FUNCTION FUN_InsideHysteresis : BOOL
VAR_INPUT
	rAct		:LREAL;			// Actual value
	rSp			:LREAL;			// Setpoint value
	rHys		:LREAL;			// Hysteresis	
END_VAR
VAR
	bInside		:BOOL;			// True if actual value is within setpoint plus minus hysteresis value
END_VAR


// Compare actual value with setpoint and hysteresis limit
IF rAct >= (rSP-rHys) AND rACT <= (rSP+rHys) THEN
	// Inside hysteresis limit
	bInside := TRUE;
ELSE
	// Outside hysteresis limit
	bInside := FALSE;
END_IF

// Set return value
FUN_InsideHysteresis := bInside;

END_FUNCTION

(* stored: Version 1.1.0.1, ProductVersion 3.1.4024.12
   POU FUN_InsideHysteresis: Id {c727d9bd-dc87-4201-b9c4-45d398efdf9d}, SpecialFunc None *)
